PROGRAM MAIN
VAR
END_VAR

Plc_Prog();

END_PROGRAM

(* stored: Version 1.1.0.1, ProductVersion 3.1.4024.9
   POU MAIN: Id {f35b5140-4c03-4eb0-96dc-6b14e615b13e}, SpecialFunc None *)
